# EPICS substitutions: iocBoot/iocMCTOptics/mctOptics.substitutions
file "$(TOP)/db/mctOptics.template"
{
pattern
{  P,      R,     CAMERA_MOTOR, LENS_MOTOR,     TOMOSCAN,       CAMERA0,  CAMERA1,      OVERLAY0,      OVERLAY1,     CAMERA_POS0, CAMERA_POS1, CAM0_LENS_POS0, CAM0_LENS_POS1, CAM0_LENS_POS2, CAM1_LENS_POS0, CAM1_LENS_POS1, CAM1_LENS_POS2, LENS_SAMPLE_X, LENS_SAMPLE_Y, LENS_SAMPLE_Z, CAM0_ROT, CAM1_ROT,  FILE_PLUGIN0,   FILE_PLUGIN1,   LENS0_FOCUS, LENS1_FOCUS,  LENS2_FOCUS, PVA_PLUGIN0,     ROI_PLUGIN0,    CB_PLUGIN0,   PVA_PLUGIN1,     ROI_PLUGIN1,    CB_PLUGIN1}
{2bm:, MCTOptics:,    2bmb:m5,    2bmb:m1,   2bmb:TomoScan:,    2bmSP1:, 2bmSP2:,  2bmSP1:Over1:,   2bmSP2:Over1:,      20,          15,     -60.030,          -0.8370,         58.64,         -60.030,        -0.8370,         58.64,        2bmb:m18,     2bmb:m57,       2bmb:m17,   2bmb:m7,  2bmb:m8,   2bmSP1:HDF1:,  2bmSP2:HDF1:,     2bmb:m2,    2bmb:m3,      2bmb:m4,   2bmSP1:Pva1:,   2bmSP1:ROI1:,  2bmSP1:CB1:, 2bmSP2:Pva1:,   2bmSP2:ROI1:,  2bmSP2:CB1:}
}
